TYPE ST_Chamber1SingleProcessCycleRecord :
STRUCT
	Result : E_Chamber1SingleProcessResult;
	FailedStage : E_Chamber1SingleProcessStage;
	FailedAxis : E_Chamber1SingleProcessAxis;
	TotalActualTime : TIME;
	StageTiming : ST_Chamber1SingleProcessStageTimings;
END_STRUCT
END_TYPE

(* stored: Version 1.1.0.1, ProductVersion 3.1.4026.18
   DUT ST_Chamber1SingleProcessCycleRecord: Id {3a36c780-9736-474d-b450-1ac197e48da4} *)
